// TIA Portal V19 export
DATA_BLOCK "HMI_IDB"   // DB45
AUTHOR : Piemme
FAMILY : System
// stored: Access Published, InstanceOfName HMI_FB, InstanceOfType FB
"HMI_FB"
   // VAR
   //    FpReadClock : Bool := FALSE;
   // END_VAR
BEGIN
END_DATA_BLOCK
